// TwinCAT 3 PLC project PLC
// ProgramVersion: 3.1.4024.0
// libraries:
//   Tc2_Standard, * (Beckhoff Automation GmbH)
//   Tc2_System, * (Beckhoff Automation GmbH)
//   Tc3_Module, * (Beckhoff Automation GmbH)
// project tree:
//   GVLs/ GVL.TcGVL
//   / PlcTask.TcTTO
//   POUs/ MAIN.TcPOU
// real-time tasks:
//   TASK PlcTask: cycle T#10ms, priority 20, ADS port 350

CONFIGURATION PLC
    RESOURCE PLC ON TwinCAT3
        TASK PlcTask(INTERVAL := T#10ms, PRIORITY := 20);
        PROGRAM MAIN WITH PlcTask : MAIN;
    END_RESOURCE
END_CONFIGURATION

// ---- GVLs/GVL.TcGVL
{attribute 'qualified_only'}
VAR_GLOBAL
	mb_Input_Coils    		: ARRAY [0..255] OF BOOL;
 	mb_Output_Coils 		: ARRAY [0..255] OF BOOL;
	
	// MB Input registers (3x) starting at address 332768
	mb_Input_Registers 		: ARRAY [0..255] OF WORD;
	
	// MB holding registers (4x) starting at address 432768
	mb_Output_Registers		: ARRAY [0..255] OF WORD;
END_VAR

// ---- POUs/MAIN.TcPOU
PROGRAM MAIN
VAR
	fbTon			: TON;
	i				: INT;
	rand			: ARRAY[0..2] OF DRAND;
	
	bAlarms			: ARRAY[0..4] OF BOOL;
	iAnalogValue	: DINT;
END_VAR

fbTon(IN:=NOT fbTon.Q, PT:=T#3S);
IF fbTon.Q THEN
	FOR i := 0 TO 2 DO
		rand[i](Seed:=i);
		GVL.mb_Input_Registers[i] := TO_WORD(rand[i].Num * 1000);
		GVL.mb_Output_Registers[i] := TO_WORD(rand[i].Num * 777);
	END_FOR
END_IF

END_PROGRAM
